// SIMATIC S7-200 project (STEP 7-Micro/WIN), CPU 224XP REL 02.01

SYMBOL_TABLE USUARIO1
PARO_1           I0.0
PARO_2           I0.1
MARCHA_1         I0.2
MARCHA_2         I0.3
LAMPARA          Q0.0
END_SYMBOL_TABLE

ORGANIZATION_BLOCK PRINCIPAL:OB1
TITLE=COMENTARIOS DEL PROGRAMA
BEGIN
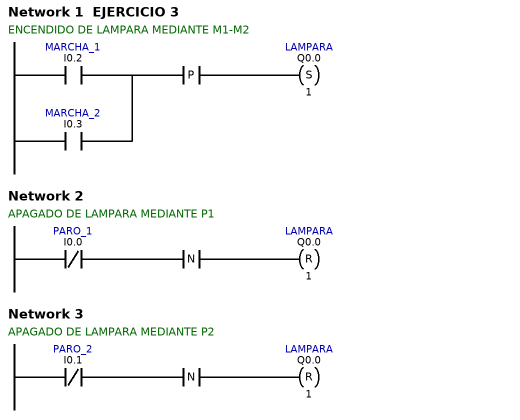
Network 1 // EJERCICIO 3
// ENCENDIDO DE LAMPARA MEDIANTE M1-M2
LD     MARCHA_1:I0.2
O      MARCHA_2:I0.3
EU
S      LAMPARA:Q0.0, 1
Network 2
// APAGADO DE LAMPARA MEDIANTE P1
LDN    PARO_1:I0.0
ED
R      LAMPARA:Q0.0, 1
Network 3
// APAGADO DE LAMPARA MEDIANTE P2
LDN    PARO_2:I0.1
ED
R      LAMPARA:Q0.0, 1
END_ORGANIZATION_BLOCK
